EventTableTriggerIO 8243: IOValue=[1], IRC5Controller=? -1, Operator=0, SignalSource=ALab_CellC_v1.0_4 5362
EventTableActionIO 8244: IOValue=[0], IRC5Controller=? -1, SignalTarget=ALab_CellC_v1.0_4 5362
EventTableEntry 8245: Group=, Trigger=conv1_buffer_upper_go_down 8246, Actions=[conv1_pallet_lifter_upper_up 8247], Comment=, ActivationMode=2, Cyclic=false
EventTableTriggerIO 8246: IOValue=[0], IRC5Controller=? -1, Operator=0, SignalSource=ALab_CellC_v1.0_4 5362
EventTableActionIO 8247: IOValue=[1], IRC5Controller=? -1, SignalTarget=ALab_CellC_v1.0_4 5362
EventTableEntry 8248: Group=, Trigger=conv1_buffer_upper_go_down 8249, Actions=[conv1_pallet_lifter_upper_down 8250], Comment=, ActivationMode=2, Cyclic=false
EventTableTriggerIO 8249: IOValue=[0], IRC5Controller=? -1, Operator=0, SignalSource=ALab_CellC_v1.0_4 5362
EventTableActionIO 8250: IOValue=[0], IRC5Controller=? -1, SignalTarget=ALab_CellC_v1.0_4 5362
EventTableEntry 8251: Group=, Trigger=conv1_buffer_upper_go_down 8252, Actions=[conv1_pallet_lifter_upper_down 8253], Comment=, ActivationMode=2, Cyclic=false
EventTableTriggerIO 8252: IOValue=[1], IRC5Controller=? -1, Operator=0, SignalSource=ALab_CellC_v1.0_4 5362
EventTableActionIO 8253: IOValue=[1], IRC5Controller=? -1, SignalTarget=ALab_CellC_v1.0_4 5362
EventTableEntry 8254: Group=, Trigger=conv1_buffer_lower_go_up 8255, Actions=[conv1_pallet_lifter_lower_down 8256], Comment=, ActivationMode=2, Cyclic=false
EventTableTriggerIO 8255: IOValue=[0], IRC5Controller=? -1, Operator=0, SignalSource=ALab_CellC_v1.0_4 5362
EventTableActionIO 8256: IOValue=[1], IRC5Controller=? -1, SignalTarget=ALab_CellC_v1.0_4 5362
EventTableEntry 8257: Group=, Trigger=conv1_buffer_lower_go_up 8258, Actions=[conv1_pallet_lifter_lower_down 8259], Comment=, ActivationMode=2, Cyclic=false
EventTableTriggerIO 8258: IOValue=[1], IRC5Controller=? -1, Operator=0, SignalSource=ALab_CellC_v1.0_4 5362
EventTableActionIO 8259: IOValue=[0], IRC5Controller=? -1, SignalTarget=ALab_CellC_v1.0_4 5362
EventTableEntry 8260: Group=, Trigger=conv2_buffer_horizontal_move 8261, Actions=[conv2_pallet_lifter_in 8262], Comment=, ActivationMode=2, Cyclic=false
EventTableTriggerIO 8261: IOValue=[1], IRC5Controller=? -1, Operator=0, SignalSource=ALab_CellC_v1.0_4 5362
EventTableActionIO 8262: IOValue=[1], IRC5Controller=? -1, SignalTarget=ALab_CellC_v1.0_4 5362
EventTableEntry 8263: Group=, Trigger=conv2_buffer_horizontal_move 8264, Actions=[conv2_pallet_lifter_in 8265], Comment=, ActivationMode=2, Cyclic=false
EventTableTriggerIO 8264: IOValue=[0], IRC5Controller=? -1, Operator=0, SignalSource=ALab_CellC_v1.0_4 5362
EventTableActionIO 8265: IOValue=[0], IRC5Controller=? -1, SignalTarget=ALab_CellC_v1.0_4 5362
EventTableEntry 8266: Group=, Trigger=conv2_buffer_horizontal_move 8267, Actions=[conv2_pallet_lifter_out 8268], Comment=, ActivationMode=2, Cyclic=false
EventTableTriggerIO 8267: IOValue=[0], IRC5Controller=? -1, Operator=0, SignalSource=ALab_CellC_v1.0_4 5362
EventTableActionIO 8268: IOValue=[1], IRC5Controller=? -1, SignalTarget=ALab_CellC_v1.0_4 5362
EventTableEntry 8269: Group=, Trigger=conv2_buffer_horizontal_move 8270, Actions=[conv2_pallet_lifter_out 8271], Comment=, ActivationMode=2, Cyclic=false
EventTableTriggerIO 8270: IOValue=[1], IRC5Controller=? -1, Operator=0, SignalSource=ALab_CellC_v1.0_4 5362
EventTableActionIO 8271: IOValue=[0], IRC5Controller=? -1, SignalTarget=ALab_CellC_v1.0_4 5362
EventTableEntry 8272: Group=, Trigger=conv2_buffer_lower_vertical_move 8273, Actions=[conv2_pallet_lifter_lower_down 8274], Comment=, ActivationMode=2, Cyclic=false
EventTableTriggerIO 8273: IOValue=[1], IRC5Controller=? -1, Operator=0, SignalSource=ALab_CellC_v1.0_4 5362
EventTableActionIO 8274: IOValue=[0], IRC5Controller=? -1, SignalTarget=ALab_CellC_v1.0_4 5362
EventTableEntry 8275: Group=, Trigger=conv2_buffer_lower_vertical_move 8276, Actions=[conv2_pallet_lifter_lower_down 8277], Comment=, ActivationMode=2, Cyclic=false
EventTableTriggerIO 8276: IOValue=[0], IRC5Controller=? -1, Operator=0, SignalSource=ALab_CellC_v1.0_4 5362
EventTableActionIO 8277: IOValue=[1], IRC5Controller=? -1, SignalTarget=ALab_CellC_v1.0_4 5362
EventTableEntry 8278: Group=, Trigger=conv2_buffer_upper_vertical_move 8279, Actions=[conv2_pallet_lifter_upper_up 8280], Comment=, ActivationMode=2, Cyclic=false
EventTableTriggerIO 8279: IOValue=[0], IRC5Controller=? -1, Operator=0, SignalSource=ALab_CellC_v1.0_4 5362
EventTableActionIO 8280: IOValue=[1], IRC5Controller=? -1, SignalTarget=ALab_CellC_v1.0_4 5362
EventTableEntry 8281: Group=, Trigger=conv2_buffer_upper_vertical_move 8282, Actions=[conv2_pallet_lifter_upper_up 8283], Comment=, ActivationMode=2, Cyclic=false
EventTableTriggerIO 8282: IOValue=[1], IRC5Controller=? -1, Operator=0, SignalSource=ALab_CellC_v1.0_4 5362
EventTableActionIO 8283: IOValue=[0], IRC5Controller=? -1, SignalTarget=ALab_CellC_v1.0_4 5362
EventTableEntry 8284: Group=, Trigger=conv2_buffer_upper_vertical_move 8285, Actions=[conv2_pallet_lifter_upper_down 8286], Comment=, ActivationMode=2, Cyclic=false
EventTableTriggerIO 8285: IOValue=[1], IRC5Controller=? -1, Operator=0, SignalSource=ALab_CellC_v1.0_4 5362
EventTableActionIO 8286: IOValue=[1], IRC5Controller=? -1, SignalTarget=ALab_CellC_v1.0_4 5362
EventTableEntry 8287: Group=, Trigger=conv2_buffer_upper_vertical_move 8288, Actions=[conv2_pallet_lifter_upper_down 8289], Comment=, ActivationMode=2, Cyclic=false
EventTableTriggerIO 8288: IOValue=[0], IRC5Controller=? -1, Operator=0, SignalSource=ALab_CellC_v1.0_4 5362
EventTableActionIO 8289: IOValue=[0], IRC5Controller=? -1, SignalTarget=ALab_CellC_v1.0_4 5362
EventTableTriggerIO 8290: IOValue=[-1], IRC5Controller=? -1, Operator=0, SignalSource=LCFA_profile 1
EventTableTriggerLogic 8291: layoutX=22, layoutY=19, Operand1=conv2_buffer_horizontal_move 8292, Operand2=? -1, Operator=2, Delay=1000
EventTableTriggerIO 8292: IOValue=[-1], IRC5Controller=? -1, Operator=0, SignalSource=ALab_CellC_v1.0_4 5362
EventTableEntry 8293: Group=, Trigger=pallet1.1 8294, Actions=[pickpallet4 8295], Comment=, ActivationMode=2, Cyclic=false
EventTableTriggerIO 8294: IOValue=[1], IRC5Controller=? -1, Operator=0, SignalSource=LCFA_profile 1
EventTableActionIO 8295: IOValue=[0], IRC5Controller=? -1, SignalTarget=LCFA_profile 1
EventTableEntry 8296: Group=, Trigger=pallet1.1 8297, Actions=[Pallet2.6 8298], Comment=, ActivationMode=2, Cyclic=false
EventTableTriggerIO 8297: IOValue=[1], IRC5Controller=? -1, Operator=0, SignalSource=LCFA_profile 1
EventTableActionIO 8298: IOValue=[0], IRC5Controller=? -1, SignalTarget=LCFA_profile 1
EventTableTriggerLogic 8357: layoutX=167, layoutY=76, Operand1=AND 4076, Operand2=AND 4081, Operator=0, Delay=1000
EventTableTriggerLogic 8358: layoutX=194, layoutY=70, Operand1=AND 4088, Operand2=AND 4093, Operator=0, Delay=1000
EventTableTriggerLogic 8359: layoutX=181, layoutY=88, Operand1=AND 4100, Operand2=AND 4105, Operator=0, Delay=1000
EventTableTriggerLogic 8360: layoutX=165, layoutY=70, Operand1=AND 4112, Operand2=AND 4117, Operator=0, Delay=1000
EventTableTriggerLogic 8361: layoutX=217, layoutY=77, Operand1=AND 4123, Operand2=AND 4127, Operator=0, Delay=1000
EventTableTriggerLogic 8362: layoutX=168, layoutY=84, Operand1=AND 4135, Operand2=AND 4139, Operator=0, Delay=1000
EventTableTriggerLogic 8363: layoutX=219, layoutY=73, Operand1=AND 4146, Operand2=AND 4150, Operator=0, Delay=1000
EventTableTriggerLogic 8364: layoutX=203, layoutY=67, Operand1=AND 4157, Operand2=AND 4161, Operator=0, Delay=1000
EventTableTriggerLogic 8365: layoutX=220, layoutY=69, Operand1=AND 4167, Operand2=AND 4171, Operator=0, Delay=1000
EventTableTriggerLogic 8366: layoutX=243, layoutY=55, Operand1=AND 4179, Operand2=AND 4183, Operator=0, Delay=1000
EventTableTriggerLogic 8367: layoutX=204, layoutY=112, Operand1=AND 4190, Operand2=AND 4194, Operator=0, Delay=1000
EventTableTriggerLogic 8368: layoutX=245, layoutY=97, Operand1=AND 4201, Operand2=AND 4205, Operator=0, Delay=1000
EventTableTriggerLogic 8369: layoutX=234, layoutY=61, Operand1=AND 4211, Operand2=AND 4214, Operator=0, Delay=1000
EventTableTriggerLogic 8370: layoutX=192, layoutY=87, Operand1=AND 4222, Operand2=AND 4225, Operator=0, Delay=1000
EventTableTriggerLogic 8371: layoutX=212, layoutY=64, Operand1=AND 4232, Operand2=AND 4235, Operator=0, Delay=1000
EventTableTriggerLogic 8372: layoutX=160, layoutY=73, Operand1=AND 4242, Operand2=AND 4245, Operator=0, Delay=1000
EventTableTriggerLogic 8373: layoutX=153, layoutY=73, Operand1=AND 4264, Operand2=NOT 4269, Operator=0, Delay=1000
EventTableTriggerLogic 8374: layoutX=133, layoutY=81, Operand1=AND 4274, Operand2=conv1_buffer_upper_go_down 6332, Operator=0, Delay=1000
EventTableTriggerLogic 8375: layoutX=184, layoutY=91, Operand1=AND 4283, Operand2=NOT 4287, Operator=0, Delay=1000
EventTableTriggerLogic 8376: layoutX=211, layoutY=90, Operand1=AND 4292, Operand2=conv1_buffer_upper_go_down 6282, Operator=0, Delay=1000
EventTableTriggerLogic 8377: layoutX=226, layoutY=110, Operand1=AND 4300, Operand2=NOT 4304, Operator=0, Delay=1000
EventTableTriggerLogic 8378: layoutX=164, layoutY=68, Operand1=AND 4309, Operand2=conv1_buffer_upper_go_down 6288, Operator=0, Delay=1000
EventTableTriggerLogic 8379: layoutX=161, layoutY=63, Operand1=AND 4317, Operand2=NOT 4320, Operator=0, Delay=1000
EventTableTriggerLogic 8380: layoutX=174, layoutY=87, Operand1=AND 4325, Operand2=conv1_buffer_upper_go_down 6294, Operator=0, Delay=1000
EventTableTriggerLogic 8381: layoutX=148, layoutY=98, Operand1=AND 4332, Operand2=NOT 4337, Operator=0, Delay=1000
EventTableTriggerLogic 8382: layoutX=206, layoutY=74, Operand1=AND 4342, Operand2=conv2_buffer_upper_vertical_move 6300, Operator=0, Delay=1000
EventTableTriggerLogic 8383: layoutX=195, layoutY=82, Operand1=AND 4351, Operand2=NOT 4355, Operator=0, Delay=1000
EventTableTriggerLogic 8384: layoutX=193, layoutY=94, Operand1=AND 4360, Operand2=conv2_buffer_upper_vertical_move 6306, Operator=0, Delay=1000
EventTableTriggerLogic 8385: layoutX=210, layoutY=27, Operand1=conv2_buffer_horizontal_move 6309, Operand2=AND 4369, Operator=0, Delay=1000
EventTableTriggerLogic 8386: layoutX=233, layoutY=95, Operand1=AND 4377, Operand2=conv2_buffer_upper_vertical_move 6312, Operator=0, Delay=1000
EventTableTriggerLogic 8387: layoutX=102, layoutY=69, Operand1=AND 4385, Operand2=NOT 4388, Operator=0, Delay=1000
EventTableTriggerLogic 8388: layoutX=97, layoutY=92, Operand1=AND 4393, Operand2=conv2_buffer_upper_vertical_move 6318, Operator=0, Delay=1000
EventTableTriggerLogic 8389: layoutX=96, layoutY=16, Operand1=cellC_pallet_holder 7125, Operand2=cellC_pallet_stopper 7126, Operator=0, Delay=1000
EventTableTriggerLogic 8390: layoutX=142, layoutY=32, Operand1=NOT 7128, Operand2=cellC_pallet_stopper 7127, Operator=0, Delay=1000
EventTableTriggerLogic 8391: layoutX=51, layoutY=46, Operand1=NOT 7130, Operand2=NOT 7132, Operator=0, Delay=1000
EventTableTriggerLogic 8392: layoutX=107, layoutY=60, Operand1=cellC_pallet_holder 7134, Operand2=NOT 7135, Operator=0, Delay=1000
EventTableTriggerIO 8394: IOValue=[1], IRC5Controller=? -1, Operator=0, SignalSource=ALab_CellC_v1.0_4 5362
EventTableTriggerLogic 8407: layoutX=184, layoutY=128, Operand1=AND 6402, Operand2=AND 6408, Operator=0, Delay=1000
EventTableTriggerLogic 8408: layoutX=231, layoutY=144, Operand1=AND 6416, Operand2=pallet1 6426, Operator=0, Delay=1000
EventTableTriggerLogic 8409: layoutX=251, layoutY=143, Operand1=AND 8115, Operand2=pallet3.1 8114, Operator=0, Delay=1000
EventTableTriggerLogic 8410: layoutX=62, layoutY=38, Operand1=pallet2 8126, Operand2=cellC_slider_horizontal_move 8125, Operator=0, Delay=1000
EventTableTriggerLogic 8411: layoutX=133, layoutY=37, Operand1=pallet3 6451, Operand2=pose6 6452, Operator=0, Delay=1000
EventTableTriggerLogic 8412: layoutX=61, layoutY=50, Operand1=pallet3.2 6456, Operand2=pose3 6457, Operator=0, Delay=1000
EventTableTriggerLogic 8413: layoutX=131, layoutY=52, Operand1=pickpallet1 6461, Operand2=pose7 6462, Operator=0, Delay=1000
EventTableTriggerLogic 8414: layoutX=8, layoutY=16, Operand1=pickpallet2 6466, Operand2=pose13 6467, Operator=0, Delay=1000
EventTableTriggerLogic 8415: layoutX=232, layoutY=117, Operand1=AND 6471, Operand2=pallet4 6481, Operator=0, Delay=1000
EventTableTriggerLogic 8416: layoutX=237, layoutY=122, Operand1=AND 6485, Operand2=conv2_buffer_stopper 6492, Operator=0, Delay=1000
EventTableTriggerLogic 8417: layoutX=240, layoutY=90, Operand1=AND 6496, Operand2=AND 6500, Operator=0, Delay=1000
EventTableTriggerLogic 8418: layoutX=80, layoutY=49, Operand1=pallet5.1 6513, Operand2=conv2_outer_lifter 6514, Operator=0, Delay=1000
EventTableTriggerIO 8419: IOValue=[1], IRC5Controller=? -1, Operator=0, SignalSource=LCFA_profile 1
EventTableTriggerIO 8420: IOValue=[1], IRC5Controller=? -1, Operator=0, SignalSource=LCFA_profile 1
EventTableTriggerIO 8421: IOValue=[1], IRC5Controller=? -1, Operator=0, SignalSource=LCFA_profile 1
EventTableTriggerIO 8422: IOValue=[1], IRC5Controller=? -1, Operator=0, SignalSource=LCFA_profile 1
EventTableTriggerIO 8423: IOValue=[1], IRC5Controller=? -1, Operator=0, SignalSource=LCFA_profile 1
EventTableTriggerIO 8424: IOValue=[1], IRC5Controller=? -1, Operator=0, SignalSource=LCFA_profile 1
EventTableTriggerIO 8425: IOValue=[1], IRC5Controller=? -1, Operator=0, SignalSource=LCFA_profile 1
EventTableTriggerIO 8426: IOValue=[1], IRC5Controller=? -1, Operator=0, SignalSource=LCFA_profile 1
EventTableTriggerIO 8427: IOValue=[1], IRC5Controller=? -1, Operator=0, SignalSource=LCFA_profile 1
EventTableTriggerIO 8428: IOValue=[1], IRC5Controller=? -1, Operator=0, SignalSource=LCFA_profile 1
EventTableTriggerIO 8429: IOValue=[0], IRC5Controller=? -1, Operator=0, SignalSource=ALab_CellC_v1.0_4 5362
EventTableTriggerIO 8430: IOValue=[1], IRC5Controller=? -1, Operator=0, SignalSource=ALab_CellC_v1.0_4 5362
EventTableTriggerIO 8431: IOValue=[0], IRC5Controller=? -1, Operator=0, SignalSource=ALab_CellC_v1.0_4 5362
EventTableTriggerIO 8432: IOValue=[1], IRC5Controller=? -1, Operator=0, SignalSource=ALab_CellC_v1.0_4 5362
EventTableTriggerIO 8433: IOValue=[1], IRC5Controller=? -1, Operator=0, SignalSource=ALab_CellC_v1.0_4 5362
EventTableTriggerIO 8434: IOValue=[0], IRC5Controller=? -1, Operator=0, SignalSource=ALab_CellC_v1.0_4 5362
EventTableTriggerIO 8435: IOValue=[0], IRC5Controller=? -1, Operator=0, SignalSource=ALab_CellC_v1.0_4 5362
EventTableTriggerIO 8436: IOValue=[1], IRC5Controller=? -1, Operator=0, SignalSource=ALab_CellC_v1.0_4 5362
EventTableTriggerIO 8437: IOValue=[1], IRC5Controller=? -1, Operator=0, SignalSource=ALab_CellC_v1.0_4 5362
EventTableTriggerIO 8438: IOValue=[0], IRC5Controller=? -1, Operator=0, SignalSource=ALab_CellC_v1.0_4 5362
EventTableTriggerIO 8439: IOValue=[1], IRC5Controller=? -1, Operator=0, SignalSource=ALab_CellC_v1.0_4 5362
EventTableTriggerIO 8440: IOValue=[0], IRC5Controller=? -1, Operator=0, SignalSource=ALab_CellC_v1.0_4 5362
EventTableTriggerIO 8441: IOValue=[0], IRC5Controller=? -1, Operator=0, SignalSource=ALab_CellC_v1.0_4 5362
EventTableTriggerIO 8442: IOValue=[1], IRC5Controller=? -1, Operator=0, SignalSource=ALab_CellC_v1.0_4 5362
EventTableTriggerIO 8443: IOValue=[1], IRC5Controller=? -1, Operator=0, SignalSource=ALab_CellC_v1.0_4 5362
EventTableTriggerIO 8444: IOValue=[0], IRC5Controller=? -1, Operator=0, SignalSource=ALab_CellC_v1.0_4 5362
EventTableTriggerIO 8445: IOValue=[0], IRC5Controller=? -1, Operator=0, SignalSource=ALab_CellC_v1.0_4 5362
EventTableTriggerIO 8446: IOValue=[1], IRC5Controller=? -1, Operator=0, SignalSource=ALab_CellC_v1.0_4 5362
EventTableTriggerIO 8447: IOValue=[1], IRC5Controller=? -1, Operator=0, SignalSource=ALab_CellC_v1.0_4 5362
EventTableTriggerIO 8448: IOValue=[0], IRC5Controller=? -1, Operator=0, SignalSource=ALab_CellC_v1.0_4 5362
EventTableTriggerIO 8449: IOValue=[1], IRC5Controller=? -1, Operator=0, SignalSource=LCFA_profile 1
EventTableTriggerIO 8450: IOValue=[1], IRC5Controller=? -1, Operator=0, SignalSource=LCFA_profile 1
EventTableTriggerIO 8451: IOValue=[1], IRC5Controller=? -1, Operator=0, SignalSource=LCFA_profile 1
EventTableTriggerIO 8452: IOValue=[1], IRC5Controller=? -1, Operator=0, SignalSource=LCFA_profile 1
EventTableTriggerIO 8453: IOValue=[1], IRC5Controller=? -1, Operator=0, SignalSource=ALab_CellC_v1.0_4 5362
EventTableTriggerIO 8454: IOValue=[0], IRC5Controller=? -1, Operator=0, SignalSource=ALab_CellC_v1.0_4 5362
EventTableTriggerIO 8455: IOValue=[1], IRC5Controller=? -1, Operator=0, SignalSource=LCFA_profile 1
EventTableTriggerIO 8456: IOValue=[1], IRC5Controller=? -1, Operator=0, SignalSource=LCFA_profile 1
EventTableTriggerIO 8457: IOValue=[1], IRC5Controller=? -1, Operator=0, SignalSource=LCFA_profile 1
EventTableTriggerIO 8458: IOValue=[1], IRC5Controller=? -1, Operator=0, SignalSource=LCFA_profile 1
EventTableTriggerIO 8459: IOValue=[1], IRC5Controller=? -1, Operator=0, SignalSource=ALab_CellC_v1.0_4 5362
EventTableTriggerIO 8460: IOValue=[0], IRC5Controller=? -1, Operator=0, SignalSource=ALab_CellC_v1.0_4 5362
EventTableTriggerIO 8461: IOValue=[1], IRC5Controller=? -1, Operator=0, SignalSource=ALab_CellC_v1.0_4 5362
EventTableTriggerIO 8462: IOValue=[0], IRC5Controller=? -1, Operator=0, SignalSource=ALab_CellC_v1.0_4 5362
EventTableTriggerIO 8463: IOValue=[0], IRC5Controller=? -1, Operator=0, SignalSource=ALab_CellC_v1.0_4 5362
EventTableTriggerIO 8464: IOValue=[1], IRC5Controller=? -1, Operator=0, SignalSource=ALab_CellC_v1.0_4 5362
EventTableTriggerIO 8465: IOValue=[1], IRC5Controller=? -1, Operator=0, SignalSource=ALab_CellC_v1.0_4 5362
EventTableTriggerIO 8466: IOValue=[0], IRC5Controller=? -1, Operator=0, SignalSource=ALab_CellC_v1.0_4 5362
EventTableTriggerIO 8471: IOValue=[1], IRC5Controller=? -1, Operator=0, SignalSource=LCFA_profile 1
EventTableTriggerIO 8472: IOValue=[1], IRC5Controller=? -1, Operator=0, SignalSource=LCFA_profile 1
EventTableTriggerIO 8473: IOValue=[1], IRC5Controller=? -1, Operator=0, SignalSource=LCFA_profile 1
EventTableTriggerLogic 8474: layoutX=150, layoutY=90, Operand1=AND 6770, Operand2=conv2_motor_s1 6766, Operator=0, Delay=1000
EventTableTriggerIO 8475: IOValue=[1], IRC5Controller=? -1, Operator=0, SignalSource=LCFA_profile 1
EventTableTriggerIO 8476: IOValue=[1], IRC5Controller=? -1, Operator=0, SignalSource=LCFA_profile 1
EventTableTriggerIO 8477: IOValue=[1], IRC5Controller=? -1, Operator=0, SignalSource=LCFA_profile 1
EventTableTriggerIO 8478: IOValue=[1], IRC5Controller=? -1, Operator=0, SignalSource=LCFA_profile 1
EventTableTriggerIO 8479: IOValue=[1], IRC5Controller=? -1, Operator=0, SignalSource=LCFA_profile 1
EventTableTriggerIO 8480: IOValue=[1], IRC5Controller=? -1, Operator=0, SignalSource=LCFA_profile 1
EventTableTriggerIO 8481: IOValue=[1], IRC5Controller=? -1, Operator=0, SignalSource=LCFA_profile 1
EventTableTriggerIO 8482: IOValue=[1], IRC5Controller=? -1, Operator=0, SignalSource=LCFA_profile 1
EventTableTriggerIO 8483: IOValue=[1], IRC5Controller=? -1, Operator=0, SignalSource=LCFA_profile 1
EventTableTriggerIO 8484: IOValue=[1], IRC5Controller=? -1, Operator=0, SignalSource=LCFA_profile 1
EventTableTriggerIO 8485: IOValue=[1], IRC5Controller=? -1, Operator=0, SignalSource=LCFA_profile 1
EventTableTriggerIO 8486: IOValue=[1], IRC5Controller=? -1, Operator=0, SignalSource=LCFA_profile 1
EventTableTriggerLogic 8487: layoutX=155, layoutY=137, Operand1=AND 6751, Operand2=NOT 6755, Operator=0, Delay=1000
EventTableTriggerIO 8488: IOValue=[1], IRC5Controller=? -1, Operator=0, SignalSource=LCFA_profile 1
EventTableTriggerIO 8489: IOValue=[1], IRC5Controller=? -1, Operator=0, SignalSource=LCFA_profile 1
EventTableTriggerLogic 8490: layoutX=48, layoutY=41, Operand1=pallet1.1 6778, Operand2=PalletIO00 6779, Operator=0, Delay=1000
EventTableTriggerIO 8491: IOValue=[1], IRC5Controller=? -1, Operator=0, SignalSource=LCFA_profile 1
EventTableTriggerIO 8492: IOValue=[1], IRC5Controller=? -1, Operator=0, SignalSource=ALab_CellC_v1.0_4 5362
EventTableTriggerIO 8493: IOValue=[0], IRC5Controller=? -1, Operator=0, SignalSource=ALab_CellC_v1.0_4 5362
EventTableTriggerLogic 8494: layoutX=103, layoutY=47, Operand1=NOT 8291, Operand2=pallet5 8290, Operator=0, Delay=1000
EventTableTriggerLogic 8495: layoutX=79, layoutY=37, Operand1=Pallet5.3 8029, Operand2=conv2_buffer_upper_vertical_move 8133, Operator=0, Delay=1000
EventTableTriggerLogic 8496: layoutX=40, layoutY=37, Operand1=Pallet5.4 8035, Operand2=conv2_buffer_lower_vertical_move 8036, Operator=0, Delay=1000
EventTableTriggerLogic 8497: layoutX=103, layoutY=47, Operand1=conv2_buffer_horizontal_move 8134, Operand2=Pallet5.7 8040, Operator=0, Delay=1000
EventTableTriggerLogic 8498: layoutX=54, layoutY=45, Operand1=NOT 8135, Operand2=Pallet5.6 8046, Operator=0, Delay=1000
EventTableTriggerLogic 8499: layoutX=108, layoutY=46, Operand1=NOT 8052, Operand2=Pallet5.5 8051, Operator=0, Delay=1000
EventTableTriggerIO 8500: IOValue=[1], IRC5Controller=? -1, Operator=0, SignalSource=LCFA_profile 1
EventTableTriggerIO 8501: IOValue=[1], IRC5Controller=? -1, Operator=0, SignalSource=LCFA_profile 1
EventTableTriggerIO 8502: IOValue=[1], IRC5Controller=? -1, Operator=0, SignalSource=LCFA_profile 1
EventTableTriggerIO 8503: IOValue=[1], IRC5Controller=? -1, Operator=0, SignalSource=LCFA_profile 1
EventTableTriggerIO 8504: IOValue=[1], IRC5Controller=? -1, Operator=0, SignalSource=LCFA_profile 1
EventTableTriggerIO 8505: IOValue=[1], IRC5Controller=? -1, Operator=0, SignalSource=LCFA_profile 1
EventTableTriggerIO 8506: IOValue=[1], IRC5Controller=? -1, Operator=0, SignalSource=LCFA_profile 1
EventTableTriggerIO 8507: IOValue=[1], IRC5Controller=? -1, Operator=0, SignalSource=LCFA_profile 1
EventTableTriggerIO 8508: IOValue=[1], IRC5Controller=? -1, Operator=0, SignalSource=LCFA_profile 1
EventTableTriggerIO 8509: IOValue=[1], IRC5Controller=? -1, Operator=0, SignalSource=LCFA_profile 1
EventTableTriggerIO 8510: IOValue=[1], IRC5Controller=? -1, Operator=0, SignalSource=LCFA_profile 1
EventTableTriggerIO 8511: IOValue=[1], IRC5Controller=? -1, Operator=0, SignalSource=LCFA_profile 1
EventTableTriggerIO 8512: IOValue=[1], IRC5Controller=? -1, Operator=0, SignalSource=LCFA_profile 1
EventTableTriggerIO 8513: IOValue=[1], IRC5Controller=? -1, Operator=0, SignalSource=LCFA_profile 1
EventTableTriggerIO 8514: IOValue=[1], IRC5Controller=? -1, Operator=0, SignalSource=LCFA_profile 1
EventTableTriggerIO 8515: IOValue=[1], IRC5Controller=? -1, Operator=0, SignalSource=LCFA_profile 1
EventTableTriggerIO 8516: IOValue=[1], IRC5Controller=? -1, Operator=0, SignalSource=LCFA_profile 1
EventTableTriggerLogic 8517: layoutX=99, layoutY=32, Operand1=Pallet2.1 8141, Operand2=NOT 8139, Operator=0, Delay=1000
EventTableTriggerLogic 8518: layoutX=181, layoutY=52, Operand1=conv1_buffer_upper_go_down 8146, Operand2=Pallet2.2 8145, Operator=0, Delay=1000
EventTableTriggerLogic 8519: layoutX=48, layoutY=51, Operand1=Pallet2.3 8150, Operand2=conv1_buffer_lower_go_up 8151, Operator=0, Delay=1000
EventTableTriggerLogic 8520: layoutX=67, layoutY=33, Operand1=pallet2 8155, Operand2=NOT 8156, Operator=0, Delay=1000
EventTableTriggerLogic 8521: layoutX=102, layoutY=29, Operand1=Pallet2.4 8161, Operand2=NOT 8162, Operator=0, Delay=1000
EventTableTriggerLogic 8522: layoutX=102, layoutY=23, Operand1=Pallet2.5 8167, Operand2=NOT 8168, Operator=0, Delay=1000
EventTableTriggerIO 8523: IOValue=[1], IRC5Controller=? -1, Operator=0, SignalSource=LCFA_profile 1
EventTableTriggerIO 8524: IOValue=[1], IRC5Controller=? -1, Operator=0, SignalSource=LCFA_profile 1
EventTableTriggerIO 8525: IOValue=[1], IRC5Controller=? -1, Operator=0, SignalSource=LCFA_profile 1
EventTableTriggerIO 8526: IOValue=[1], IRC5Controller=? -1, Operator=0, SignalSource=LCFA_profile 1
EventTableTriggerIO 8527: IOValue=[1], IRC5Controller=? -1, Operator=0, SignalSource=LCFA_profile 1
EventTableTriggerIO 8528: IOValue=[1], IRC5Controller=? -1, Operator=0, SignalSource=LCFA_profile 1
EventTableTriggerIO 8529: IOValue=[1], IRC5Controller=? -1, Operator=0, SignalSource=LCFA_profile 1
EventTableTriggerIO 8530: IOValue=[1], IRC5Controller=? -1, Operator=0, SignalSource=LCFA_profile 1
EventTableTriggerIO 8531: IOValue=[1], IRC5Controller=? -1, Operator=0, SignalSource=LCFA_profile 1
EventTableTriggerIO 8532: IOValue=[1], IRC5Controller=? -1, Operator=0, SignalSource=LCFA_profile 1
EventTableTriggerIO 8533: IOValue=[1], IRC5Controller=? -1, Operator=0, SignalSource=LCFA_profile 1
EventTableTriggerIO 8534: IOValue=[1], IRC5Controller=? -1, Operator=0, SignalSource=LCFA_profile 1
EventTableTriggerIO 8535: IOValue=[1], IRC5Controller=? -1, Operator=0, SignalSource=LCFA_profile 1
EventTableTriggerLogic 8536: layoutX=49, layoutY=26, Operand1=Pallet2.6 8213, Operand2=conv1_buffer_horizontal_open 8214, Operator=0, Delay=1000
EventTableTriggerIO 8537: IOValue=[1], IRC5Controller=? -1, Operator=0, SignalSource=LCFA_profile 1
EventTableTriggerIO 8538: IOValue=[1], IRC5Controller=? -1, Operator=0, SignalSource=LCFA_profile 1
EventTableTriggerIO 8539: IOValue=[1], IRC5Controller=? -1, Operator=0, SignalSource=LCFA_profile 1
EventTableTriggerIO 8540: IOValue=[1], IRC5Controller=? -1, Operator=0, SignalSource=LCFA_profile 1
EventTableTriggerIO 8541: IOValue=[1], IRC5Controller=? -1, Operator=0, SignalSource=LCFA_profile 1
EventTableTriggerIO 8542: IOValue=[1], IRC5Controller=? -1, Operator=0, SignalSource=ALab_CellC_v1.0_4 5362
EventTableTriggerIO 8543: IOValue=[0], IRC5Controller=? -1, Operator=0, SignalSource=ALab_CellC_v1.0_4 5362
EventTableTriggerIO 8544: IOValue=[1], IRC5Controller=? -1, Operator=0, SignalSource=ALab_CellC_v1.0_4 5362
EventTableTriggerIO 8545: IOValue=[0], IRC5Controller=? -1, Operator=0, SignalSource=ALab_CellC_v1.0_4 5362
EventTableTriggerIO 8546: IOValue=[1], IRC5Controller=? -1, Operator=0, SignalSource=ALab_CellC_v1.0_4 5362
EventTableTriggerIO 8547: IOValue=[0], IRC5Controller=? -1, Operator=0, SignalSource=ALab_CellC_v1.0_4 5362
EventTableTriggerIO 8548: IOValue=[0], IRC5Controller=? -1, Operator=0, SignalSource=ALab_CellC_v1.0_4 5362
EventTableTriggerIO 8549: IOValue=[1], IRC5Controller=? -1, Operator=0, SignalSource=ALab_CellC_v1.0_4 5362
EventTableTriggerIO 8550: IOValue=[0], IRC5Controller=? -1, Operator=0, SignalSource=ALab_CellC_v1.0_4 5362
EventTableTriggerIO 8551: IOValue=[1], IRC5Controller=? -1, Operator=0, SignalSource=ALab_CellC_v1.0_4 5362
EventTableTriggerIO 8552: IOValue=[1], IRC5Controller=? -1, Operator=0, SignalSource=ALab_CellC_v1.0_4 5362
EventTableTriggerIO 8553: IOValue=[0], IRC5Controller=? -1, Operator=0, SignalSource=ALab_CellC_v1.0_4 5362
EventTableTriggerIO 8554: IOValue=[0], IRC5Controller=? -1, Operator=0, SignalSource=ALab_CellC_v1.0_4 5362
EventTableTriggerIO 8555: IOValue=[1], IRC5Controller=? -1, Operator=0, SignalSource=ALab_CellC_v1.0_4 5362
EventTableTriggerIO 8556: IOValue=[1], IRC5Controller=? -1, Operator=0, SignalSource=ALab_CellC_v1.0_4 5362
EventTableTriggerIO 8557: IOValue=[0], IRC5Controller=? -1, Operator=0, SignalSource=ALab_CellC_v1.0_4 5362
EventTableTriggerIO 8558: IOValue=[0], IRC5Controller=? -1, Operator=0, SignalSource=ALab_CellC_v1.0_4 5362
EventTableTriggerIO 8559: IOValue=[1], IRC5Controller=? -1, Operator=0, SignalSource=ALab_CellC_v1.0_4 5362
EventTableTriggerIO 8560: IOValue=[1], IRC5Controller=? -1, Operator=0, SignalSource=ALab_CellC_v1.0_4 5362
EventTableTriggerIO 8561: IOValue=[0], IRC5Controller=? -1, Operator=0, SignalSource=ALab_CellC_v1.0_4 5362
EventTableTriggerIO 8562: IOValue=[1], IRC5Controller=? -1, Operator=0, SignalSource=LCFA_profile 1
EventTableTriggerIO 8563: IOValue=[1], IRC5Controller=? -1, Operator=0, SignalSource=LCFA_profile 1
EventTableEntry 8586: Group=, Trigger=Rob1_Gripper_set 8587, Actions=[EventTableActionMechanicalPose 8588], Comment=, ActivationMode=2, Cyclic=false
EventTableTriggerIO 8587: IOValue=[1], IRC5Controller=? -1, Operator=0, SignalSource=ALab_CellC_v1.0_4 5362
EventTableActionMechanicalPose 8588: VirtualSignal=, Mechanism=Gripper 8576, ToPoseName=ClosePose, VirtualSignalValue=[1]
EventTableEntry 8589: Group=, Trigger=Rob1_Gripper_set 8590, Actions=[EventTableActionMechanicalPose 8591], Comment=, ActivationMode=2, Cyclic=false
EventTableTriggerIO 8590: IOValue=[0], IRC5Controller=? -1, Operator=0, SignalSource=ALab_CellC_v1.0_4 5362
EventTableActionMechanicalPose 8591: VirtualSignal=, Mechanism=Gripper 8576, ToPoseName=ClosePose, VirtualSignalValue=[1]
EventTableEntry 8592: Group=, Trigger=Rob1_Gripper_reset 8593, Actions=[EventTableActionMechanicalPose 8594], Comment=, ActivationMode=2, Cyclic=false
EventTableTriggerIO 8593: IOValue=[1], IRC5Controller=? -1, Operator=0, SignalSource=ALab_CellC_v1.0_4 5362
EventTableActionMechanicalPose 8594: VirtualSignal=, Mechanism=Gripper 8576, ToPoseName=HomePosition, VirtualSignalValue=[1]
EventTableEntry 8595: Group=, Trigger=Rob1_Gripper_reset 8596, Actions=[EventTableActionMechanicalPose 8597], Comment=, ActivationMode=2, Cyclic=false
EventTableTriggerIO 8596: IOValue=[0], IRC5Controller=? -1, Operator=0, SignalSource=ALab_CellC_v1.0_4 5362
EventTableActionMechanicalPose 8597: VirtualSignal=, Mechanism=Gripper 8576, ToPoseName=HomePosition, VirtualSignalValue=[1]
Station logic (signal -> signal, property => property):
  ALab_CellC_v1.0_4.Rob1_Gripper_Reset -> Rubic Cube Simulation .DI_Open
  ALab_CellC_v1.0_4.Rob1_Gripper_Set -> Rubic Cube Simulation .DI_Close
Targets, tools, work objects and paths stored in the station and not in the controller backup, written as RAPID:
! task T_ROB2
MODULE CalibData
  TASK PERS wobjdata Wobjmytool:=[TRUE,TRUE,"",[[0,0,0],[1,0,0,0]],[[0,0,0],[1,0,0,0]]];
ENDMODULE


--- Backups/ALab_CellC_v1.0_4/RAPID/TASK1/PROGMOD/CalibData.mod ---
MODULE CalibData
    PERS tooldata Gripper_1:=[TRUE,[[0,0,50],[1,0,0,0]],[1,[0,0,1],[1,0,0,0],0,0,0]];
ENDMODULE

--- Backups/ALab_CellC_v1.0_4/RAPID/TASK1/PROGMOD/MainModule.mod ---
MODULE MainModule

    PROC main()
        HomePosition;

        ! Value "1" sets on the Digital Output
        ! Value "0" sets off the Digital Output

        SetDO Rob1_Gripper_Reset,1;
        SetDO Rob1_Gripper_Reset,0;
        WaitTime 1;
        SetDO Rob1_Gripper_Set,1;
        SetDO Rob1_Gripper_Set,0;

    ENDPROC

    PROC HomePosition()
		MoveAbsJ [[0,0,0,0,0,0],[9E9,9E9,9E9,9E9,9E9,9E9]]\NoEOffs,v200,z50,tool0;
	ENDPROC
ENDMODULE

--- Backups/ALab_CellC_v1.0_4/SYSPAR/EIO.cfg ---
EIO:CFG_1.0:5:0::
#
EIO_BUS:

      -Name "Virtual1" -ConnectorID "SIM1"

      -Name "DeviceNet1" -BusType "DNET" -ConnectorID "PCI1"\
      -ConnectorLabel "First DeviceNet"

      -Name "DeviceNet2" -BusType "DNET" -ConnectorID "PCI2"\
      -ConnectorLabel "Second DeviceNet" -DN_MasterAddress 1
#
EIO_UNIT_TYPE:

      -Name "Virtual" -VendorName "ABB" -ProductName "Virtual unit"

      -Name "DN_GENERIC" -BusType "DNET" -DN_ExplicitMsgEnabled \
      -DN_C1OutputSize -1 -DN_C1InputSize -1

      -Name "d320" -BusType "DNET" -VendorName "ABB Robotics"\
      -ProductName "120 Vac Unit" -DN_VendorId 75 -DN_ProductCode 1\
      -DN_DeviceType 7 -DN_MajorRev 1 -DN_ExplicitMsgEnabled  -DN_C1Interval 50\
      -DN_C1OutputSize 2 -DN_C1InputSize 2

      -Name "d327" -BusType "DNET" -VendorName "ABB Robotics"\
      -ProductName "Combi Unit" -DN_VendorId 75 -DN_ProductCode 2\
      -DN_DeviceType 100 -DN_MajorRev 5 -DN_ExplicitMsgEnabled \
      -DN_C1Interval 50 -DN_C1OutputSize 6 -DN_C1InputSize 2

      -Name "d328" -BusType "DNET" -VendorName "ABB Robotics"\
      -ProductName "24 VDC Unit" -DN_VendorId 75 -DN_ProductCode 3\
      -DN_DeviceType 7 -DN_ExplicitMsgEnabled  -DN_C1Interval 50\
      -DN_C1OutputSize 2 -DN_C1InputSize 2

      -Name "d332" -BusType "DNET" -VendorName "ABB Robotics"\
      -ProductName "Relay Unit" -DN_VendorId 75 -DN_ProductCode 5\
      -DN_DeviceType 7 -DN_MajorRev 2 -DN_ExplicitMsgEnabled  -DN_C1Interval 50\
      -DN_C1OutputSize 2 -DN_C1InputSize 2

      -Name "d327A" -BusType "DNET" -VendorName "ABB Robotics"\
      -ProductName "Combi Unit" -DN_VendorId 75 -DN_ProductCode 2\
      -DN_DeviceType 100 -DN_MajorRev 5 -DN_ExplicitMsgEnabled  -DN_C1Type "COS"\
      -DN_C1OutputSize 6 -DN_C1InputSize 2

      -Name "d328A" -BusType "DNET" -VendorName "ABB Robotics"\
      -ProductName "24 VDC Unit" -DN_VendorId 75 -DN_ProductCode 3\
      -DN_DeviceType 7 -DN_ExplicitMsgEnabled  -DN_C1Type "COS"\
      -DN_C1OutputSize 2 -DN_C1InputSize 2

      -Name "d332A" -BusType "DNET" -VendorName "ABB Robotics"\
      -ProductName "Relay Unit" -DN_VendorId 75 -DN_ProductCode 5\
      -DN_DeviceType 7 -DN_MajorRev 2 -DN_ExplicitMsgEnabled  -DN_C1Type "COS"\
      -DN_C1OutputSize 2 -DN_C1InputSize 2

      -Name "d355A" -BusType "DNET" -VendorName "ABB Robotics"\
      -ProductName "Analog Unit" -DN_VendorId 75 -DN_ProductCode 10\
      -DN_DeviceType 100 -DN_MajorRev 1 -DN_ExplicitMsgEnabled \
      -DN_C1Interval 50 -DN_C1OutputSize 8 -DN_C1InputSize 8

      -Name "d651" -BusType "DNET" -VendorName "ABB Robotics"\
      -ProductName "Combi Unit" -DN_VendorId 75 -DN_ProductCode 25\
      -DN_DeviceType 100 -DN_ExplicitMsgEnabled  -DN_C1Type "COS"\
      -DN_C1OutputSize 5 -DN_C1InputSize 1

      -Name "d652" -BusType "DNET" -VendorName "ABB Robotics"\
      -ProductName "24 VDC Unit" -DN_VendorId 75 -DN_ProductCode 26\
      -DN_DeviceType 7 -DN_ExplicitMsgEnabled  -DN_C1Type "COS"\
      -DN_C1OutputSize 2 -DN_C1InputSize 2

      -Name "d653" -BusType "DNET" -VendorName "ABB Robotics"\
      -ProductName "Relay Unit" -DN_VendorId 75 -DN_ProductCode 27\
      -DN_DeviceType 7 -DN_ExplicitMsgEnabled  -DN_C1Type "COS"\
      -DN_C1OutputSize 1 -DN_C1InputSize 1

      -Name "DN_SLAVE" -BusType "DNET" -DN_VendorId 8 -DN_ProductCode 12\
      -DN_DeviceType 12 -DN_ExplicitMsgEnabled  -DN_C1Interval 50\
      -DN_C1OutputSize 8 -DN_C1InputSize 8

      -Name "S4CPLUS_DN_SLAVE" -BusType "DNET" -DN_VendorId 75\
      -DN_ProductCode 15 -DN_DeviceType 100 -DN_C1Interval 50\
      -DN_C1OutputSize 22 -DN_C1InputSize 22

      -Name "d350A" -BusType "DNET" -VendorName "ABB Robotics"\
      -ProductName "RIO Adapter" -DN_VendorId 75 -DN_ProductCode 6\
      -DN_DeviceType 7 -DN_MajorRev 2 -DN_ExplicitMsgEnabled  -DN_C1Type "COS"\
      -DN_C1OutputSize -1 -DN_C1InputSize -1

      -Name "d351A" -BusType "DNET" -VendorName "ABB Robotics"\
      -ProductName "IBS Adapter" -DN_VendorId 75 -DN_ProductCode 7\
      -DN_DeviceType 7 -DN_MajorRev 1 -DN_ExplicitMsgEnabled  -DN_C1Type "COS"\
      -DN_C1OutputSize -1 -DN_C1InputSize -1

      -Name "d352A" -BusType "DNET" -VendorName "ABB Robotics"\
      -ProductName "PBUS Adapter" -DN_VendorId 75 -DN_ProductCode 8\
      -DN_DeviceType 7 -DN_MajorRev 1 -DN_ExplicitMsgEnabled  -DN_C1Type "COS"\
      -DN_C1OutputSize -1 -DN_C1InputSize -1

      -Name "d378A" -BusType "DNET" -VendorName "ABB Robotics"\
      -ProductName "CCLink Adapter" -DN_VendorId 75 -DN_ProductCode 17\
      -DN_DeviceType 7 -DN_MajorRev 1 -DN_ExplicitMsgEnabled \
      -DN_C1OutputSize -1 -DN_C1InputSize -1

      -Name "DN_omron_drt2_xwt" -BusType "DNET" -VendorName "drt_xwt"\
      -DN_VendorId 47 -DN_DeviceType 7 -DN_C1OutputSize -1 -DN_C1InputSize -1

      -Name "DN_smc_pneumatics" -BusType "DNET" -VendorName "ex120-sdn1"\
      -DN_VendorId 7 -DN_DeviceType 16 -DN_C1OutputSize -1 -DN_C1InputSize -1

      -Name "DN_BECKHOFF" -BusType "DNET" -VendorName "Beckhoff"\
      -ProductName "LC4200" -DN_VendorId 134 -DN_ProductCode 5200\
      -DN_DeviceType 12
#
EIO_UNIT:

      -Name "DN_conv2" -UnitType "DN_omron_drt2_xwt" -Bus "DeviceNet1"\
      -DN_Address 13

      -Name "DN_conv1" -UnitType "DN_omron_drt2_xwt" -Bus "DeviceNet1"\
      -DN_Address 12

      -Name "DN_conv2_pneumatics" -UnitType "DN_smc_pneumatics"\
      -Bus "DeviceNet1" -DN_Address 17

      -Name "DN_conv1_pneumatics" -UnitType "DN_smc_pneumatics"\
      -Bus "DeviceNet1" -DN_Address 16

      -Name "DN_cell_c" -UnitType "DN_omron_drt2_xwt" -Bus "DeviceNet1"\
      -DN_Address 14

      -Name "DN_cell_pneumatics" -UnitType "DN_smc_pneumatics" -Bus "DeviceNet1"\
      -DN_Address 18

      -Name "Local_DeviceNet" -UnitType "d332A" -Bus "DeviceNet1"\
      -UnitLabel "For user interface and doors" -DN_Address 10

      -Name "DN_robo1" -UnitType "DN_GENERIC" -Bus "DeviceNet2"\
      -UnitLabel "DNrobo1" -DN_Address 21

      -Name "DN_robo2" -UnitType "DN_GENERIC" -Bus "DeviceNet2"\
      -UnitLabel "DNrobo2" -DN_Address 27
#
EIO_SIGNAL:

      -Name "conv1_pallet_out" -SignalType "DI" -Unit "DN_conv1" -UnitMap "00"

      -Name "conv1_pallet_buffer" -SignalType "DI" -Unit "DN_conv1"\
      -UnitMap "01"

      -Name "conv1_pallet_lifter_in" -SignalType "DI" -Unit "DN_conv1"\
      -UnitMap "04"

      -Name "conv1_pallet_lifter_out" -SignalType "DI" -Unit "DN_conv1"\
      -UnitMap "05"

      -Name "conv1_pallet_lifter_lower_down" -SignalType "DI" -Unit "DN_conv1"\
      -UnitMap "06"

      -Name "conv1_pallet_lifter_upper_up" -SignalType "DI" -Unit "DN_conv1"\
      -UnitMap "07"

      -Name "conv1_pallet_lifter_upper_down" -SignalType "DI" -Unit "DN_conv1"\
      -UnitMap "08"

      -Name "conv1_outer_lifter_down" -SignalType "DI" -Unit "DN_conv1"\
      -UnitMap "09"

      -Name "conv1_outer_lifter_up" -SignalType "DI" -Unit "DN_conv1"\
      -UnitMap "10"

      -Name "conv1_buffer_upper_go_down" -SignalType "DO"\
      -Unit "DN_conv1_pneumatics" -SignalLabel "0 = up" -UnitMap "2"

      -Name "conv1_buffer_horizontal_open" -SignalType "DO"\
      -Unit "DN_conv1_pneumatics" -SignalLabel "0 = close" -UnitMap "0"

      -Name "conv1_buffer_lower_go_up" -SignalType "DO"\
      -Unit "DN_conv1_pneumatics" -SignalLabel "0 = down" -UnitMap "4"

      -Name "conv1_outer_lifter" -SignalType "DO" -Unit "DN_conv1_pneumatics"\
      -SignalLabel "0 = up" -UnitMap "6"

      -Name "conv2_pallet_out" -SignalType "DI" -Unit "DN_conv2" -UnitMap "00"

      -Name "conv2_pallet_buffer" -SignalType "DI" -Unit "DN_conv2"\
      -UnitMap "02"

      -Name "conv2_middle_up_sensor" -SignalType "DI" -Unit "DN_conv2"\
      -UnitMap "03"

      -Name "conv2_pallet_lifter_in" -SignalType "DI" -Unit "DN_conv2"\
      -UnitMap "04"

      -Name "conv2_pallet_lifter_out" -SignalType "DI" -Unit "DN_conv2"\
      -UnitMap "05"

      -Name "conv2_pallet_lifter_upper_down" -SignalType "DI" -Unit "DN_conv2"\
      -UnitMap "06"

      -Name "conv2_pallet_lifter_upper_up" -SignalType "DI" -Unit "DN_conv2"\
      -UnitMap "07"

      -Name "conv2_pallet_lifter_lower_down" -SignalType "DI" -Unit "DN_conv2"\
      -UnitMap "08"

      -Name "conv2_outer_lifter_down" -SignalType "DI" -Unit "DN_conv2"\
      -UnitMap "09"

      -Name "conv2_outer_lifter_up" -SignalType "DI" -Unit "DN_conv2"\
      -UnitMap "10"

      -Name "conv2_pallet_stopper_up" -SignalType "DI" -Unit "DN_conv2"\
      -UnitMap "11"

      -Name "conv2_pallet_stopper_down" -SignalType "DI" -Unit "DN_conv2"\
      -UnitMap "12"

      -Name "conv2_something_fiberopt" -SignalType "DI" -Unit "DN_conv2"\
      -UnitMap "13"

      -Name "conv2_buffer_stopper" -SignalType "DO" -Unit "DN_conv2_pneumatics"\
      -SignalLabel "1 = stop" -UnitMap "8"

      -Name "conv2_buffer_upper_vertical_move" -SignalType "DO"\
      -Unit "DN_conv2_pneumatics" -SignalLabel "0 = up" -UnitMap "2"

      -Name "conv2_buffer_lower_vertical_move" -SignalType "DO"\
      -Unit "DN_conv2_pneumatics" -SignalLabel "0 = down" -UnitMap "4"

      -Name "conv2_outer_lifter" -SignalType "DO" -Unit "DN_conv2_pneumatics"\
      -SignalLabel "0 = up" -UnitMap "6"

      -Name "conv2_buffer_horizontal_move" -SignalType "DO"\
      -Unit "DN_conv2_pneumatics" -SignalLabel "0 = close" -UnitMap "0"

      -Name "System_air_release" -SignalType "DO" -Unit "DN_conv1_pneumatics"\
      -SignalLabel "1 = release" -UnitMap " 8"

      -Name "cellC_slider_horizontal_move" -SignalType "DO"\
      -Unit "DN_cell_pneumatics" -SignalLabel "0 = top of conv1" -UnitMap " 0"

      -Name "cellC_slider_vertical_move" -SignalType "DO"\
      -Unit "DN_cell_pneumatics" -SignalLabel "0 = up" -UnitMap "2"

      -Name "cellC_gripper_horizontal_move" -SignalType "DO"\
      -Unit "DN_cell_pneumatics" -SignalLabel "0 = close" -UnitMap "4"

      -Name "cellC_gripper_vertical_move" -SignalType "DO"\
      -Unit "DN_cell_pneumatics" -SignalLabel "0 = close" -UnitMap "6"

      -Name "cellC_pallet_stopper" -SignalType "DO" -Unit "DN_cell_pneumatics"\
      -SignalLabel "0 = stop" -UnitMap "8"

      -Name "cellC_pallet_holder" -SignalType "DO" -Unit "DN_cell_pneumatics"\
      -SignalLabel "0 = hold" -UnitMap "10"

      -Name "conv1_motor_s1" -SignalType "DO" -Unit "DN_conv1"\
      -SignalLabel "motor forward/STOP" -UnitMap "00" -SysfailReset

      -Name "conv1_motor_s2" -SignalType "DO" -Unit "DN_conv1"\
      -SignalLabel "motor STOP/reverse" -UnitMap "01"

      -Name "conv1_motor_s5" -SignalType "DO" -Unit "DN_conv1"\
      -SignalLabel "motor acceleration" -UnitMap " 02"

      -Name "conv2_motor_s1" -SignalType "DO" -Unit "DN_conv2"\
      -SignalLabel "motor forward/STOP" -UnitMap "00" -SysfailReset

      -Name "conv2_motor_s2" -SignalType "DO" -Unit "DN_conv2"\
      -SignalLabel "motor STOP/reverse" -UnitMap "01"

      -Name "conv2_motor_s5" -SignalType "DO" -Unit "DN_conv2"\
      -SignalLabel "motor acceleration" -UnitMap "02"

      -Name "cellC_pallet_conv1" -SignalType "DI" -Unit "DN_cell_c"\
      -UnitMap "00"

      -Name "cellC_pallet_conv2" -SignalType "DI" -Unit "DN_cell_c"\
      -UnitMap "01"

      -Name "cellC_02" -SignalType "DI" -Unit "DN_cell_c" -UnitMap "02"

      -Name "cellC_03" -SignalType "DI" -Unit "DN_cell_c" -UnitMap "03"

      -Name "cellC_slider_over_conv2" -SignalType "DI" -Unit "DN_cell_c"\
      -UnitMap "04"

      -Name "cellC_slider_over_conv1" -SignalType "DI" -Unit "DN_cell_c"\
      -UnitMap "05"

      -Name "cellC_slider_down" -SignalType "DI" -Unit "DN_cell_c" -UnitMap "06"

      -Name "cellC_slider_up" -SignalType "DI" -Unit "DN_cell_c" -UnitMap "07"

      -Name "cellC_gripper_horizontal_closed" -SignalType "DI" -Unit "DN_cell_c"\
      -UnitMap "08"

      -Name "cellC_gripper_vertical_open" -SignalType "DI" -Unit "DN_cell_c"\
      -UnitMap "09"

      -Name "cellC_stopper_closed" -SignalType "DI" -Unit "DN_cell_c"\
      -UnitMap "10"

      -Name "cellC_stopper_open" -SignalType "DI" -Unit "DN_cell_c"\
      -UnitMap "11"

      -Name "cellC_pallet_holder_closed" -SignalType "DI" -Unit "DN_cell_c"\
      -UnitMap "12"

      -Name "cellC_pallet_holder_open" -SignalType "DI" -Unit "DN_cell_c"\
      -UnitMap "13"

      -Name "UI_KOTIASEMAPYYNTO" -SignalType "DI" -Unit "Local_DeviceNet"\
      -SignalLabel "Initial state" -UnitMap "00"

      -Name "UI_SEIS" -SignalType "DI" -Unit "Local_DeviceNet"\
      -SignalLabel "Stop" -UnitMap "01"

      -Name "UI_KAYNTIIN" -SignalType "DI" -Unit "Local_DeviceNet"\
      -SignalLabel "Start" -UnitMap "02"

      -Name "UI_VIRHEKUITTAUS" -SignalType "DI" -Unit "Local_DeviceNet"\
      -SignalLabel "Reset" -UnitMap "03"

      -Name "UI_NAYTEPYYNTO" -SignalType "DI" -Unit "Local_DeviceNet"\
      -SignalLabel "Sample" -UnitMap "04"

      -Name "UI_ALOITUSAJO" -SignalType "DI" -Unit "Local_DeviceNet"\
      -SignalLabel "System in run mode" -UnitMap "05"

      -Name "TestPlateDrive" -SignalType "DO" -Unit "Local_DeviceNet"\
      -SignalLabel "0 = out, 1 = in" -UnitMap "05"

      -Name "SecurityLightYellow" -SignalType "DO" -Unit "Local_DeviceNet"\
      -UnitMap "06"

      -Name "SecurityLightRed" -SignalType "DO" -Unit "Local_DeviceNet"\
      -UnitMap "07"

      -Name "SecurityLightWhite" -SignalType "DO" -Unit "Local_DeviceNet"\
      -UnitMap "08"

      -Name "Light_NAYTEPYYNTO" -SignalType "DO" -Unit "Local_DeviceNet"\
      -UnitMap "04"

      -Name "Light_VIRHEKUITTAUS" -SignalType "DO" -Unit "Local_DeviceNet"\
      -UnitMap "03"

      -Name "Light_KAYNTIIN" -SignalType "DO" -Unit "Local_DeviceNet"\
      -UnitMap "02"

      -Name "Light_SEIS" -SignalType "DO" -Unit "Local_DeviceNet" -UnitMap "01"

      -Name "Light_KOTIASEMAPYYNTO" -SignalType "DO" -Unit "Local_DeviceNet"\
      -UnitMap "00"

      -Name "Rob1_Gripper_Set" -SignalType "DO" -Unit "DN_robo1" -UnitMap "6"\
      -Access "ALL"

      -Name "Rob1_Gripper_Reset" -SignalType "DO" -Unit "DN_robo1" -UnitMap "7"\
      -Access "ALL"

      -Name "Rob2_Gripper_Reset" -SignalType "DO" -Unit "DN_robo2" -UnitMap "7"\
      -Access "ALL"

      -Name "Rob2_Gripper_Set" -SignalType "DO" -Unit "DN_robo2" -UnitMap "6"\
      -Access "ALL"
#
EIO_COMMAND_TYPE:

      -Name "LinkAddr" -UnitType "d350A" -DefValue "1" -OrderNr 1\
      -DN_Path "6,20 64 24 01 30 01,C6,1"

      -Name "DataRate" -UnitType "d350A" -DefValue "0" -OrderNr 2\
      -DN_Path "6,20 64 24 01 30 02,C6,1"

      -Name "StartQ" -UnitType "d350A" -DefValue "0" -OrderNr 3\
      -DN_Path "6,20 64 24 01 30 03,C6,1"

      -Name "RackSize" -UnitType "d350A" -DefValue "0" -OrderNr 4\
      -DN_Path "6,20 64 24 01 30 04,C6,1"

      -Name "LastRack" -UnitType "d350A" -DefValue "0" -OrderNr 5\
      -DN_Path "6,20 64 24 01 30 05,C1,1"

      -Name "D350Areset" -UnitType "d350A" -DefValue "0" -OrderNr 6\
      -DN_Path "4,20 01 24 01,C1,1" -DN_Service 5

      -Name "DataWidth" -UnitType "d351A" -DefValue "3" -OrderNr 1\
      -DN_Path "6,20 65 24 01 30 01,C6,1"

      -Name "D351Areset" -UnitType "d351A" -DefValue "0" -OrderNr 2\
      -DN_Path "4,20 01 24 01,C1,1" -DN_Service 5

      -Name "MasterInputSize" -UnitType "d352A" -DefValue "1" -OrderNr 1\
      -DN_Path "6,20 67 24 01 30 02,C6,1"

      -Name "MasterOutputSize" -UnitType "d352A" -DefValue "1" -OrderNr 2\
      -DN_Path "6,20 67 24 01 30 03,C6,1"

      -Name "StationAddress" -UnitType "d352A" -DefValue "126" -OrderNr 3\
      -DN_Path "6,20 67 24 01 30 04,C6,1"

      -Name "D352Areset" -UnitType "d352A" -DefValue "0" -OrderNr 4\
      -DN_Path "4,20 01 24 01,C1,1" -DN_Service 5

      -Name "StationNo" -UnitType "d378A" -DefValue "1" -OrderNr 1\
      -DN_Path "6,20 68 24 01 30 01,C6,1"

      -Name "BaudRate" -UnitType "d378A" -DefValue "0" -OrderNr 2\
      -DN_Path "6,20 68 24 01 30 02,C6,1"

      -Name "OccStat" -UnitType "d378A" -DefValue "1" -OrderNr 3\
      -DN_Path "6,20 68 24 01 30 03,C6,1"

      -Name "BasicIO" -UnitType "d378A" -DefValue "0" -OrderNr 4\
      -DN_Path "6,20 68 24 01 30 04,C1,1"

      -Name "D378Areset" -UnitType "d378A" -DefValue "0" -OrderNr 5\
      -DN_Path "4,20 01 24 01,C1,1" -DN_Service 5
#
EIO_ACCESS:

      -Name "ALL" -Rapid  -LocalManual  -LocalAuto  -RemoteManual  -RemoteAuto
